// TIA Portal V17 export
// export: Created 2022-07-28T18:03:03.3888611Z, ExportSetting None, DisplayName Totally Integrated Automation Portal, DisplayVersion V17, DisplayName TIA Portal Openness, DisplayVersion V17, DisplayName TIA Portal Teamcenter Gateway, DisplayVersion V17, DisplayName TIA Portal Version Control Interface, DisplayVersion V17, DisplayName TIA Portal Test Suite Advanced, DisplayVersion V17, DisplayName SINAMICS Startdrive Advanced, DisplayVersion V17, DisplayName SINAMICS DCC, DisplayVersion V17, DisplayName SINAMICS Startdrive G130, G150, S120, S150, SINAMICS MV, S210, DisplayVersion V17, DisplayName SINAMICS Startdrive G110M, G120, G120C, G120D, G120P, G115D, DisplayVersion V17, DisplayName STEP 7 Professional, DisplayVersion V17, DisplayName SIMATIC Energy Suite, DisplayVersion V17, DisplayName STEP 7 CFC, DisplayVersion V17, DisplayName STEP 7 Safety, DisplayVersion V17, DisplayName WinCC Advanced / Unified PC, DisplayVersion V17, DisplayName SIMATIC Visualization Architect, DisplayVersion V17
DATA_BLOCK "D_PLC_CTRL"   // DB7
// stored: InstanceOfName Lib_FB_PLC, InstanceOfType FB
"Lib_FB_PLC"
   // VAR_IN_OUT
   //    IO_PLC : "Lib_UDT_PLC";
   // END_VAR
   // VAR
   //    TMBITS_PREV : Int;
   //    MEM_RUNTIME : LReal;
   //    FB_LTIME : LReal;
   //    FB_LTIME_1 : Real;
   //    TIME_TCK_ms : LReal;
   //    TIME_TCK_s : LReal;
   //    TIME_TCK_min : Real;
   //    TIME_TCK_ms_1 : DInt;
   //    TIME_TCK_ms_2 : UDInt;
   //    TIME_TCK_ms_3 : DInt;
   //    TIME_TCK_min_3rs : Real;
   //    OB1 : Struct
   //       PrevOutputTime : Date_And_Time;
   //       cyclicTime : Int;
   //    END_STRUCT;
   //    TIME_ZONE : Struct
   //       Set : Bool;
   //       DONE : Bool;
   //       BUSY : Bool;
   //       ERROR : Bool;
   //       STATUS : Word;
   //       TimeTransformationRule : TimeTransformationRule;
   //    END_STRUCT;
   //    SET_TIMEZONE_Instance { ExternalAccessible := 'False'; ExternalVisible := 'False'; ExternalWritable := 'False'} : SET_TIMEZONE;
   // END_VAR
BEGIN
END_DATA_BLOCK
